Staubli VAL3: Reset.pgx

public program Reset()
  local num l_i
begin
  //报警复位
  for l_i=0 to nAxesSum-1
    call cmdFaultReset(l_i)
  endFor
//  call user:timerDialog("复位完成",0.5)
end
